// TIA Portal V19 export
ORGANIZATION_BLOCK "MainOB"   // OB1, LAD, ProgramCycle
TITLE = "Main Program Sweep (Cycle)"
{ S7_Optimized_Access := 'TRUE' }
// stored: SetENOAutomatically false
   VAR_INPUT
      Initial_Call : Bool;   // Initial call of this OB
      Remanence : Bool;   // =True, if remanent data are available
   END_VAR
   VAR_TEMP   // added for the SCL form of the ladder/FBD networks
      _w1 : Bool;
   END_VAR
BEGIN

REGION Network 1
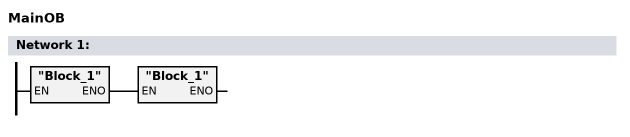
   RUNG wire#powerrail
      "Block_1"()
      "Block_1"()
   END_RUNG
   // the same network as SCL:
   "Block_1"(ENO => #_w1);
   IF #_w1 THEN "Block_1"(); END_IF;
END_REGION
END_ORGANIZATION_BLOCK
